type T_Syntax_Types :
struct
    nSubrange : int(0..100) := 50;
    aMatrix : array[1..3, 1..3] of real;
    sCustomText : string(255);
end_struct
end_type

(* stored: Version 1.1.0.1, ProductVersion 3.1.4024.16
   DUT T_Syntax_Types: Id {10e3c610-3666-4282-840d-2574b4694439} *)
